{attribute addProperty BoxType "AX8620-0000-0026"}
{attribute addProperty Id "Reserve_0BIT10.1251Ready_to_operateBIT10.1252TorqueOFF_order_nBIT10.1253Brake_ramp_order_nBIT10.1254Limit_dc_link_current_order_nBIT10.1255NC_handling_order_nBIT10.1256Counter_BIT_0BIT10.12512Counter_BIT_1BIT10.12512Counter_BIT_2BIT10.12512Counter_BIT_3BIT10.12512Counter_BIT_4BIT10.12512"}
{attribute addProperty CRC "995667025"}
{attribute addProperty SizeInBites "16"}
{attribute addProperty SizeInBytes "2"}
TYPE Statusword_3B58AC51 :
STRUCT
	{attribute addProperty Name "Reserve_0"}
	Reserve_0 : BIT;
	{attribute addProperty Name "Ready_to_operate"}
	Ready_to_operate : BIT;
	{attribute addProperty Name "TorqueOFF_order_n"}
	TorqueOFF_order_n : BIT;
	{attribute addProperty Name "Brake_ramp_order_n"}
	Brake_ramp_order_n : BIT;
	{attribute addProperty Name "Limit_dc_link_current_order_n"}
	Limit_dc_link_current_order_n : BIT;
	{attribute addProperty Name "NC_handling_order_n"}
	NC_handling_order_n : BIT;
	{attribute 'hide'}
	reserve_1_BIT_0 : BIT;
	{attribute 'hide'}
	reserve_1_BIT_1 : BIT;
	{attribute 'hide'}
	reserve_2_BIT_0 : BIT;
	{attribute 'hide'}
	reserve_2_BIT_1 : BIT;
	{attribute 'hide'}
	reserve_2_BIT_2 : BIT;
	{attribute addProperty Name "Counter"}
	Counter_BIT_0 : BIT;
	{attribute addProperty Name "Counter"}
	Counter_BIT_1 : BIT;
	{attribute addProperty Name "Counter"}
	Counter_BIT_2 : BIT;
	{attribute addProperty Name "Counter"}
	Counter_BIT_3 : BIT;
	{attribute addProperty Name "Counter"}
	Counter_BIT_4 : BIT;
END_STRUCT
END_TYPE

(* stored: Version 1.2.0.0, ProductVersion 3.1.4024.9
   DUT Statusword_3B58AC51: Id {87848566-0ed9-4354-a5f1-6fa77a4d1d4d} *)
